FUNCTION_BLOCK HeaderAccessor IMPLEMENTS I_SessionHeaderAccessor, I_ServerResponseHeaderAccessor, I_AsyncResponseHeaderAccessor, I_ChunkedResponseHeaderAccessor, I_ChunkedRequestsHeaderAccessor, I_RpcHeaderAccessor

PROPERTY PUBLIC ContentType_Json : T_MAXSTRING
GET
ContentType_Json := 'application/json';
END_GET
END_PROPERTY

PROPERTY PUBLIC HeaderKey_Accept : T_MAXSTRING
GET
HeaderKey_Accept := 'Accept';
END_GET
END_PROPERTY

PROPERTY PUBLIC HeaderKey_ChunkSequence : T_MAXSTRING
GET
HeaderKey_ChunkSequence := 'Chunk-Sequence';
END_GET
END_PROPERTY

PROPERTY PUBLIC HeaderKey_ChunkTotal : T_MAXSTRING
GET
HeaderKey_ChunkTotal := 'Chunk-Total';
END_GET
END_PROPERTY

PROPERTY PUBLIC HeaderKey_ContentType : T_MAXSTRING
GET
HeaderKey_ContentType := 'Content-Type';
END_GET
END_PROPERTY

PROPERTY PUBLIC HeaderKey_HasMoreChunks : T_MAXSTRING
GET
HeaderKey_HasMoreChunks := 'Has-More-Chunks';
END_GET
END_PROPERTY

PROPERTY PUBLIC HeaderKey_Message : T_MAXSTRING
GET
HeaderKey_Message := 'Message';
END_GET
END_PROPERTY

PROPERTY PUBLIC HeaderKey_MethodName : T_MAXSTRING
GET
HeaderKey_MethodName := 'Method-Name';
END_GET
END_PROPERTY

PROPERTY PUBLIC HeaderKey_RequestId : T_MAXSTRING
GET
HeaderKey_RequestId := 'Request-Id';
END_GET
END_PROPERTY

PROPERTY PUBLIC HeaderKey_ResponseId : T_MAXSTRING
GET
HeaderKey_ResponseId := 'Response-Id';
END_GET
END_PROPERTY

PROPERTY PUBLIC HeaderKey_RetryDelay : T_MAXSTRING
GET
HeaderKey_RetryDelay := 'Retry-Delay';
END_GET
END_PROPERTY

PROPERTY PUBLIC HeaderKey_SessionId : T_MAXSTRING
GET
HeaderKey_SessionId := 'Session-Id';
END_GET
END_PROPERTY

PROPERTY PUBLIC HeaderKey_Status : T_MAXSTRING
GET
HeaderKey_Status := 'Status';
END_GET
END_PROPERTY

PROPERTY PUBLIC HeaderKey_Type : T_MAXSTRING
GET
HeaderKey_Type := 'Type';
END_GET
END_PROPERTY

PROPERTY PUBLIC StatusValue_Accepted : T_MAXSTRING
GET
StatusValue_Accepted := 'Accepted';
END_GET
END_PROPERTY

PROPERTY PUBLIC StatusValue_Busy : T_MAXSTRING
GET
StatusValue_Busy := 'Busy';
END_GET
END_PROPERTY

PROPERTY PUBLIC StatusValue_Error : T_MAXSTRING
GET
StatusValue_Error := 'Error';
END_GET
END_PROPERTY

PROPERTY PUBLIC StatusValue_Pending : T_MAXSTRING
GET
StatusValue_Pending := 'Pending';
END_GET
END_PROPERTY

PROPERTY PUBLIC StatusValue_Success : T_MAXSTRING
GET
StatusValue_Success := 'Success';
END_GET
END_PROPERTY

METHOD PUBLIC TryGetAcceptResponseFormatFromRequest : BOOL
VAR_INPUT
	Request : I_Request;
	Destination : ANY;
END_VAR
TryGetAcceptResponseFormatFromRequest := Request.Header.TryGetField(HeaderKey_Accept,Destination);
END_METHOD

METHOD PUBLIC TryGetChunkSequenceFromRequest : BOOL
VAR_INPUT
	Request : I_Request;
	Destination : REFERENCE TO DINT;
END_VAR
VAR
	chunkSequence : DINT;
END_VAR
IF NOT Request.Header.TryGetField(HeaderKey_ChunkSequence,chunkSequence) THEN
	RETURN;
END_IF

Destination := chunkSequence;
TryGetChunkSequenceFromRequest := TRUE;
END_METHOD

METHOD PUBLIC TryGetChunkTotalFromRequest : BOOL
VAR_INPUT
	Request : I_Request;
	Destination : REFERENCE TO DINT;
END_VAR
VAR
	chunkTotal : DINT;
END_VAR
IF NOT Request.Header.TryGetField(HeaderKey_ChunkTotal,chunkTotal) THEN
	RETURN;
END_IF

Destination := chunkTotal;
TryGetChunkTotalFromRequest := TRUE;
END_METHOD

METHOD PUBLIC TryGetContentTypeFromRequest : BOOL
VAR_INPUT
	Request : I_Request;
	Destination : ANY;
END_VAR
TryGetContentTypeFromRequest := Request.Header.TryGetField(HeaderKey_ContentType,Destination);
END_METHOD

METHOD PUBLIC TryGetHasMoreChunksFromRequest : BOOL
VAR_INPUT
	Request : I_Request;
	Destination : REFERENCE TO BOOL;
END_VAR
VAR
	hasMoreChunks : BOOL;
END_VAR
IF NOT Request.Header.TryGetField(HeaderKey_HasMoreChunks,hasMoreChunks) THEN
	RETURN;
END_IF

Destination := hasMoreChunks;
TryGetHasMoreChunksFromRequest := TRUE;
END_METHOD

METHOD PUBLIC TryGetMethodNameFromRequest : BOOL
VAR_INPUT
	Request : I_Request;
	Destination : ANY;
END_VAR
TryGetMethodNameFromRequest := Request.Header.TryGetField(HeaderKey_MethodName,Destination);
END_METHOD

METHOD PUBLIC TryGetRequestIdFromRequest : BOOL
VAR_INPUT
	Request : I_Request;
	Destination : REFERENCE TO T_MAXSTRING;
END_VAR
VAR
	requestId : T_MAXSTRING;
END_VAR
IF NOT Request.Header.TryGetField(HeaderKey_RequestId,requestId) THEN
	RETURN;
END_IF

Destination := requestId;
TryGetRequestIdFromRequest := TRUE;
END_METHOD

METHOD PUBLIC TryGetResponseIdFromRequest : BOOL
VAR_INPUT
	Request : I_Request;
	Destination : ANY;
END_VAR
TryGetResponseIdFromRequest := Request.Header.TryGetField(HeaderKey_ResponseId,Destination);
END_METHOD

METHOD PUBLIC TryGetSessionIdFromRequest : BOOL
VAR_INPUT
	Request : I_Request;
	Destination : REFERENCE TO T_MAXSTRING;
END_VAR
VAR
	sessionId : T_MAXSTRING;
END_VAR
IF NOT Request.Header.TryGetField(HeaderKey_SessionId, sessionId) THEN
	RETURN;
END_IF

Destination := sessionId;
TryGetSessionIdFromRequest := TRUE;
END_METHOD

METHOD PUBLIC TryGetSessionIdFromResponse : BOOL
VAR_INPUT
	Response : I_ServerResponse;
	Destination : ANY;
END_VAR
TryGetSessionIdFromResponse := Response.Header.TryGetField(HeaderKey_SessionId,Destination);
END_METHOD

METHOD PUBLIC TryGetTypeFromRequest : BOOL
VAR_INPUT
	Request : I_Request;
	Destination : ANY;
END_VAR
TryGetTypeFromRequest := Request.Header.TryGetField(HeaderKey_Type,Destination);
END_METHOD

METHOD PUBLIC UpdateRequestWithSessionId
VAR_INPUT
	Request : I_Request;
	SessionId : T_MAXSTRING;
END_VAR
Request.Header.TryWriteField(HeaderKey_SessionId,SessionId);
END_METHOD

METHOD PUBLIC UpdateResponseWithAccepted
VAR_INPUT
	Response : I_ServerResponse;
END_VAR
VAR
	status : T_MAXSTRING; // this was needed to fix the 4026 error with using ANY and properties
END_VAR
status := StatusValue_Accepted;
Response.Header.TryWriteField(HeaderKey_Status, status);
END_METHOD

METHOD PUBLIC UpdateResponseWithBusy
VAR_INPUT
	Response : I_ServerResponse;
END_VAR
VAR
	status : T_MAXSTRING; // this was needed to fix the 4026 error with using ANY and properties
END_VAR
status := StatusValue_Busy;
Response.Header.TryWriteField(HeaderKey_Status, status);
END_METHOD

METHOD PUBLIC UpdateResponseWithError
VAR_INPUT
	Response : I_ServerResponse;
	Message : T_MAXSTRING;
END_VAR
VAR
	status : T_MAXSTRING; // this was needed to fix the 4026 error with using ANY and properties
END_VAR
status := StatusValue_Error;
Response.Header.TryWriteField(HeaderKey_Status, status);
Response.Header.TryWriteField(HeaderKey_Message, Message);
END_METHOD

METHOD PUBLIC UpdateResponseWithHasMoreChunks
VAR_INPUT
	Response : I_ServerResponse;
	ResponseId : T_MAXSTRING;
END_VAR
VAR
	hasMoreChunks : BOOL := TRUE;
END_VAR
Response.Header.TryWriteField(HeaderKey_ResponseId,ResponseId);
Response.Header.TryWriteField(HeaderKey_HasMoreChunks,hasMoreChunks);
END_METHOD

METHOD PUBLIC UpdateResponseWithPending
VAR_INPUT
	Response : I_ServerResponse;
	ResponseId : T_MAXSTRING;
	RetryDelayInMs : UDINT;
END_VAR
VAR
	retryDelayInMsString : T_MAXSTRING;
	status : T_MAXSTRING; // this was needed to fix the 4026 error with using ANY and properties
END_VAR
status := StatusValue_Pending;
Response.Header.TryWriteField(HeaderKey_Status, status);
Response.Header.TryWriteField(HeaderKey_ResponseId, ResponseId);

IF RetryDelayInMs > 0 THEN
	retryDelayInMsString := UDINT_TO_STRING(RetryDelayInMs);
	Response.Header.TryWriteField(HeaderKey_RetryDelay, retryDelayInMsString);
END_IF
END_METHOD

METHOD PUBLIC UpdateResponseWithSessionId
VAR_INPUT
	Response : I_ServerResponse;
	SessionId : T_MAXSTRING;
END_VAR
Response.Header.TryWriteField(HeaderKey_SessionId,SessionId);
END_METHOD

METHOD PUBLIC UpdateResponseWithSuccess
VAR_INPUT
	Response : I_ServerResponse;
END_VAR
VAR
	status : T_MAXSTRING; // this was needed to fix the 4026 error with using ANY and properties
END_VAR
status := StatusValue_Success;
Response.Header.TryWriteField(HeaderKey_Status, status);
END_METHOD

END_FUNCTION_BLOCK

(* stored: Version 1.1.0.1, ProductVersion 3.1.4024.13
   POU HeaderAccessor: Id {d021ecca-620e-0860-1f0e-52fe0a5ee06d}, SpecialFunc None
   Folder Constants: Id {4b76e81e-166f-07f2-2dc7-b9df2184ff4b}
   Property ContentType_Json: Id {1a546b78-c0bd-0c73-3937-e7fca9d02677}
   Get Get: Id {81db8599-9864-0db8-01c0-05e744dadd07}
   Property HeaderKey_Accept: Id {cdb44211-93bd-0f8d-1b06-b5325aeaf814}
   Get Get: Id {a6f07aa9-ac71-06ae-2700-1193207a30f6}
   Property HeaderKey_ChunkSequence: Id {cbb5c4dc-ca92-0d2b-23d0-f8f1537dec2c}
   Get Get: Id {83207506-298f-04b9-332b-4978d328baa3}
   Property HeaderKey_ChunkTotal: Id {83952441-c48b-0d75-1a3b-e1717e4fd1ce}
   Get Get: Id {2f97f3e3-aece-08a0-1c8b-c6016ad56bf4}
   Property HeaderKey_ContentType: Id {cd3b755d-cded-06de-3f03-14b6492ae3df}
   Get Get: Id {39042b97-95f8-01ce-0749-41ad8825cd2e}
   Property HeaderKey_HasMoreChunks: Id {32886e17-e83b-0acf-0d65-b901dca4cc0a}
   Get Get: Id {5cfd1418-a3b0-03e8-308f-4dbf7ccd4b57}
   Property HeaderKey_Message: Id {c473bf28-9c3d-0d16-0730-d54e3bf39f8a}
   Get Get: Id {e302caf0-03e0-0cfa-161e-a0840e8dae93}
   Property HeaderKey_MethodName: Id {00602141-973f-03c4-2a5d-e21d85a5c963}
   Get Get: Id {d8f5dc44-f08e-0b33-00a6-6739c2b52b4b}
   Property HeaderKey_RequestId: Id {3c14d5b4-65fe-01b8-3a84-e04618d2f82e}
   Get Get: Id {215d4c24-b139-061f-3be7-bd55c0ff6dc4}
   Property HeaderKey_ResponseId: Id {8002bcb8-12b6-04d7-14a2-97a5663f42e6}
   Get Get: Id {8882a1bb-7502-02f5-3195-7218d1a5d767}
   Property HeaderKey_RetryDelay: Id {27dbf177-e933-076f-2c08-641432c640be}
   Get Get: Id {ef5e8adf-96f0-0a16-193e-723171ab5134}
   Property HeaderKey_SessionId: Id {2c9bc0fe-e5ae-0d0b-1e19-b0923fe7d0c0}
   Get Get: Id {24fd20fc-73bb-0d75-1c1a-8f236a47d5de}
   Property HeaderKey_Status: Id {c0677b16-13ec-080c-1091-87890690a3d5}
   Get Get: Id {261adbaf-e250-000e-379a-6c50d4e60e01}
   Property HeaderKey_Type: Id {5009e799-257b-05d8-254d-0bfa93574a47}
   Get Get: Id {c39318b6-5fe7-0ff5-1321-08ac3c310011}
   Property StatusValue_Accepted: Id {90344a30-da2c-072e-2a3e-8edbeda51004}
   Get Get: Id {e2a993f4-1abb-06b0-1f60-88956ec70025}
   Property StatusValue_Busy: Id {cbba375a-45b6-0fe7-3f86-dbc983603351}
   Get Get: Id {73cc720d-2263-0c66-2242-ffb0d2beb88d}
   Property StatusValue_Error: Id {92fb372a-c766-04b2-082d-628e79b08852}
   Get Get: Id {aed43d11-867e-05fa-255d-201bbe0fe194}
   Property StatusValue_Pending: Id {bc06f6e0-91f6-08e7-147d-cbe398ddb90f}
   Get Get: Id {6f7891cd-3149-0c05-37bc-f40bd281e2db}
   Property StatusValue_Success: Id {c0ce3bcd-3fbf-0dc7-1772-cdaf9d48bdcc}
   Get Get: Id {0e942a4d-828f-0790-1e58-86d37f6acf65}
   Method TryGetAcceptResponseFormatFromRequest: Id {661b798b-5f89-0689-3016-67b00e4cfb9b}
   Method TryGetChunkSequenceFromRequest: Id {99c3935f-c4f8-0139-2540-10dca180a4d5}
   Method TryGetChunkTotalFromRequest: Id {124ea5ac-b697-0475-3406-63e83be8bba6}
   Method TryGetContentTypeFromRequest: Id {9e1445fd-a2e5-01ea-24c9-250d4eee359d}
   Method TryGetHasMoreChunksFromRequest: Id {bc882e48-cb84-0466-3b65-4ceb421fd8a1}
   Method TryGetMethodNameFromRequest: Id {a2520f56-2ea7-0769-345d-8a000a1bba9c}
   Method TryGetRequestIdFromRequest: Id {6033cd6f-04db-08d6-2916-1f792c890009}
   Method TryGetResponseIdFromRequest: Id {1ee9e1fa-0495-0c4f-0b0b-43f7dea31f71}
   Method TryGetSessionIdFromRequest: Id {e4307ac2-e1a4-023b-207a-f8bed391f36e}
   Method TryGetSessionIdFromResponse: Id {db4ccf79-84dc-08a1-1fb0-f9ccb3c3acdf}
   Method TryGetTypeFromRequest: Id {e7c1136e-4da5-03b4-0629-2af28771f0f8}
   Method UpdateRequestWithSessionId: Id {cee472c7-f147-0ea0-0f43-c6db452a989e}
   Method UpdateResponseWithAccepted: Id {af108ee6-d2c3-04ac-1b24-52a7ac863a46}
   Method UpdateResponseWithBusy: Id {4987f0f3-6fc2-05c5-3890-68e51493446a}
   Method UpdateResponseWithError: Id {2e898d81-f520-029c-17f5-197a713d6b2e}
   Method UpdateResponseWithHasMoreChunks: Id {d85749f5-b28e-02dd-3ee1-61d49f38421c}
   Method UpdateResponseWithPending: Id {ab48b1d8-ba64-0403-1be4-3f554a08d3cb}
   Method UpdateResponseWithSessionId: Id {2f8c81f9-7dfb-0bd3-2613-44bbaca1ca47}
   Method UpdateResponseWithSuccess: Id {6b6cb74a-5cde-07e8-23ac-7702e5c969d7} *)
